FUNCTION_BLOCK ClearLinkMC EXTENDS FBA_TrifectaDrive IMPLEMENTS I_EncodedDrive
VAR_OUTPUT
	pulse AT %Q* : INT;
	brakeRelease AT %Q* : BOOL := TRUE;
	enable : BOOL;
	A : BOOL;
	B : BOOL;
	clear : BOOL;
END_VAR
VAR	
	hlfb AT %I* : REAL := -9999; //high level feedback, if -9999 then servo is idle
	
	outputRegister AT %Q* : INT;
	pulseRequest : INT;
	
	homingDelay : TON;
	resetPulse : TP;
	
	mode : (HOLD, TARGET, CONTINUOUS, RESET_ERR);
	calculation : (IDLE, DOWN, UP, CALCULATE, DONE);
	maxPosition : LREAL;
	
	position, targetPos : LREAL;
	
	pulsePosition : INT;
	pulseCounter : INT;
	rotationsPerPulse : INT; //revolutions per pulse
	displacementPerPulse : LREAL; //displacement per pulse
END_VAR
VAR_STAT CONSTANT
	resetWidth : TIME := T#500MS;
	delayWidth : TIME := T#500MS;
END_VAR
VAR //constructor
	homingDirectionOut : BOOL; 			//homing direction - see <A>
	minPosition : LREAL;
	displacementPerRotation : LREAL; 	//displacement per revolution	
	unitsPerPulse : INT := 800; 		//800 Teknic units per rotation - default setting is 800 units (1 rotation) per pulse
END_VAR

//M-connector output register
outputRegister.0 := enable AND bEnable; 	//enable
outputRegister.1 := A; 						//direction bit - T = outwards, F = inwards
outputRegister.2 := B; 						//homing bit - after startup, set to TRUE to begin homing, then set to FALSE to finish homing
outputRegister.3 := clear; 					//reset bit

rotationsPerPulse := unitsPerPulse/800; //Teknic constant - 800 units per rotation
displacementPerPulse := displacementPerRotation * rotationsPerPulse;

resetPulse(IN:= , PT:= resetWidth, Q=> clear, ET=> ); //reset pulse

IF NOT enable AND NOT AtInnerLimit THEN
	homingComplete := FALSE;
	step := Homing.IDLE;
	mode := HOLD;
END_IF

override();

CASE mode OF		
	HOLD: //hold current position, no motion
		pulse := 0;
		pulseRequest := 0;
	
	TARGET:	//target a given position
		
		IF WithinTolerance(position, targetPos, displacementPerPulse) THEN
			pulseRequest := 0;
			pulse := 0;
			mode := HOLD;
			
		ELSIF NOT Active THEN
			A :=  position < targetPos;
			(*
			2 options to traverse to a target position:
				a)  send all pulses at once - continuous motion but may exceed limits, check for bounds before setting
				b)  1 pulse at a time - choppy but safer
			*)
			targetPos := MAX(targetPos, minPosition); //if below minPosition, set to minPosition
			targetPos := MIN(targetPos, maxPosition); //if above maxPosition, set to maxPosition
			
			pulseRequest := TO_INT(ABS(position - targetPos)/displacementPerPulse);
			//pulseRequest := 1;
		END_IF
		
	CONTINUOUS: //single pulses in the direction specified by moveContinuous()
		pulseRequest := 1;
		
	RESET_ERR: //reset pulse, servo may need to be rehomed aftewards
		pulse := 0;
		pulseRequest := 0;
		resetPulse.IN := TRUE;
		
		IF resetPulse.Q THEN
			resetPulse.IN := FALSE;
			mode := HOLD;
		END_IF
		
END_CASE

sequence();

PROPERTY Active : BOOL
GET
Active := hlfb <> -9999;
END_GET
END_PROPERTY

{attribute 'monitoring':='call'}
PROPERTY AtOuterLimit : BOOL
GET
AtOuterLimit := outerLimit <> limitSensorDefaultState;
END_GET
END_PROPERTY

METHOD PRIVATE calculatePositions : BOOL
(*
the purpose of this method is calculate the position at the outer limit

complete a full range traverse while counting the pulses, then multiply
	displacement per rotation
	rotations per pulse
	number of pulses for the traversal
and add to position at inner limit to get position at outer limit
*)
CASE calculation OF
	IDLE:
		calculation := DOWN;
		
	DOWN:
		moveContinuous(direction := MC_Negative_Direction);
		IF AtInnerLimit THEN
			calculation := UP;
			pulseCounter := 0;
		END_IF
		
	UP:
		moveContinuous(direction := MC_Positive_Direction);
		IF AtHome THEN
			maxPosition := minPosition + (displacementPerRotation * rotationsPerPulse * pulseCounter);
			calculation := DONE;
		END_IF
		
	DONE:
		calculation := 0;
		calculatePositions := TRUE;
		
END_CASE
END_METHOD

PROPERTY CurrentPosition : LREAL
GET
CurrentPosition := position;

//CurrentPosition := pulsePosition * displacementPerPulse;
END_GET
SET
position := CurrentPosition;
END_SET
END_PROPERTY

PROPERTY Error : BOOL
GET
END_GET
END_PROPERTY

METHOD homingSequence : BOOL
homingDelay(IN:= , PT:= delayWidth, Q=> , ET=> );

CASE step OF
	Homing.IDLE:
		enable := TRUE;
		A := FALSE;
		B := TRUE;
		brakeRelease := TRUE;
		
		homingComplete := FALSE;
		
		homingDelay.IN := TRUE;
		IF homingDelay.Q THEN
			homingDelay.IN := FALSE;
			//step := Homing.START;
			step := Homing.RETRY;
		END_IF
		
	Homing.START:
		IF homingDelay.Q THEN
			homingDelay.IN := FALSE;
			step := Homing.SET;
			
		ELSIF AtHome THEN
			homingDelay.IN := TRUE;
			
		ELSIF AtOuterLimit THEN
			step := Homing.RETRY;
		
		ELSE
			enable := TRUE;
			A := FALSE;
			B := TRUE;
			brakeRelease := TRUE;
		
		END_IF
	
	Homing.RETRY:
		IF AtInnerLimit THEN
			homingDelay.IN := TRUE;
			enable := FALSE;
			
			IF homingDelay.Q THEN
				homingDelay.IN := FALSE;
				step := Homing.START;
			END_IF
			
		ELSE
			enable := TRUE;
			A := FALSE;
			B := FALSE;
			brakeRelease := TRUE;
			
			mode := CONTINUOUS;
		END_IF

	Homing.SET:
		enable := TRUE;
		A := FALSE;
		B := FALSE;
		brakeRelease := TRUE;
		
		IF calculatePositions() THEN
			step := Homing.DONE;
		END_IF
		
	Homing.DONE:
		homingSequence := homingComplete := TRUE;
		
		pulsePosition := 0;
		
		mode := HOLD;
		step := Homing.IDLE;
	
END_CASE
END_METHOD

{attribute 'TcRpcEnable'}
METHOD moveAbsolute : BOOL
VAR_INPUT
	newTarget : LREAL;
END_VAR
IF target >= maxPosition AND target <= minPosition THEN
	A :=  position < targetPos;
	targetPos := newTarget;
	mode := TARGET;
	
	moveAbsolute := TRUE;
END_IF
END_METHOD

{attribute 'TcRpcEnable'}
METHOD moveContinuous : BOOL
VAR_INPUT
	direction : MC_Direction;
END_VAR
IF direction = MC_Negative_Direction THEN
	A := FALSE;
ELSIF direction = MC_Positive_Direction THEN
	A := TRUE;
END_IF

mode := CONTINUOUS;
END_METHOD

{attribute 'TcRpcEnable'}
METHOD moveRelative : BOOL
VAR_INPUT
	distance : LREAL;
END_VAR
targetPos := targetPos + distance;

mode := TARGET;
END_METHOD

METHOD PRIVATE override : BOOL
VAR_INPUT
END_VAR
(*
allowable motion is between AtHome and AtInnerLimit
*)
IF AtHome AND NOT Active THEN
	IF homingDirectionOut THEN //homing is outwards
		position := maxPosition;
		pulsePosition := pulseCounter;
	ELSE
		position := minPosition;
		pulsePosition := 0;
	END_IF
	

ELSIF AtInnerLimit AND NOT Active THEN
	IF homingDirectionOut THEN //homing is outwards
		position := minPosition;
		pulsePosition := 0;
	ELSE
		position := maxPosition;
		pulsePosition := pulseCounter;
	END_IF
END_IF

CASE mode OF		
	HOLD:
		//
	
	TARGET:
		IF
			(AtHome AND TargetPosition > CurrentPosition) OR
			(AtInnerLimit AND TargetPosition > CurrentPosition) OR
			(AtOuterLimit AND TargetPosition < CurrentPosition)
		THEN
			mode := HOLD;
		END_IF
		
	CONTINUOUS:
		IF
			(AtHome AND A) OR
			(AtInnerLimit AND A) OR
			(AtOuterLimit AND NOT A)
		THEN
			mode := HOLD;
		END_IF
		
	RESET_ERR:
		//
		
END_CASE
END_METHOD

METHOD reset : BOOL
VAR_INPUT
END_VAR
mode := RESET_ERR;
END_METHOD

METHOD PRIVATE sequence : BOOL
VAR_INPUT
END_VAR
IF Active THEN //servo is active
	IF A THEN //positive direction
		position := position + (displacementPerPulse * pulse);
		pulsePosition := pulsePosition + pulse;
		
		pulseCounter := pulseCounter + pulse;
	ELSE //negative direction
		position := position - (displacementPerPulse * pulse);
		pulsePosition := pulsePosition - pulse;
		
		pulseCounter := pulseCounter - pulse;
	END_IF
	pulse := 0; //pulses already received, can be set to 0 so position change is not compounded

ELSIF pulse = 0 THEN //servo is not active
	pulse := pulseRequest;
END_IF

pulseRequest := 0; //remove this if not working as intended
END_METHOD

METHOD stop : BOOL
VAR_INPUT
END_VAR
mode := HOLD;
END_METHOD

PROPERTY TargetPosition : LREAL
GET
END_GET
SET
targetPos := TargetPosition;
END_SET
END_PROPERTY

METHOD toHome : BOOL
VAR_INPUT
END_VAR
IF homingDirectionOut THEN
	moveAbsolute(newTarget := maxPosition);
ELSE
	moveAbsolute(newTarget := minPosition);
END_IF
END_METHOD

END_FUNCTION_BLOCK

(* stored: Version 1.1.0.1, ProductVersion 3.1.4024.11
   POU ClearLinkMC: Id {c959ba26-8558-4921-981d-1da3c299d707}, SpecialFunc None
   Folder Private: Id {9b3fea93-f350-4628-abcc-bd49e2d7cd99}
   Folder Properties: Id {e78b63fe-cf71-47b5-ba6b-3023a80b30ce}
   Property Active: Id {807c9ae6-2791-4a9b-8015-1bf451a6a56b}
   Get Get: Id {aa4cc01a-37da-43cb-b30c-8e2bc563783d}
   Property AtOuterLimit: Id {6385a979-b10d-4caf-84a5-664acfc88266}
   Get Get: Id {eb0add8c-74bc-4bc2-93ab-6fcb2fc36408}
   Method calculatePositions: Id {e19e2a50-fb22-4fdb-a61a-d177c769d547}
   Property CurrentPosition: Id {75ebdd6d-7b75-4de5-8593-621bb72d6114}
   Get Get: Id {6856d05c-951f-4e2e-87df-ebd187d24ea1}
   Set Set: Id {1fda77e3-f52e-4259-845a-7410fc523da0}
   Property Error: Id {bda12f76-8849-4aa6-a93d-2a3f2d50597e}
   Get Get: Id {fa80b17b-fc29-4649-956e-d05d2b8946f1}
   Method homingSequence: Id {ab2757a4-d5f6-4f3f-addc-5f1377a21651}
   Method moveAbsolute: Id {50ef4f22-8da2-4b4e-8432-de0919b36ac2}
   Method moveContinuous: Id {6fae7e55-36e1-434b-b1d0-5392145a2ede}
   Method moveRelative: Id {a27e0a4f-4fbc-4d22-bb40-916e67eef58b}
   Method override: Id {c88d925b-2a9b-44f5-b155-07becad1ca73}
   Method reset: Id {148910f4-ce89-4537-a99c-bb0337253006}
   Method sequence: Id {a500267c-ac9c-4314-ade9-3f5adbe892a2}
   Method stop: Id {9c245f97-172f-4533-81f7-d28245b80a16}
   Property TargetPosition: Id {46ee9331-03d8-4e80-977f-3f6ec7fad893}
   Get Get: Id {c9bb5ba2-9737-4f8b-a18e-17d189211f37}
   Set Set: Id {b9e464bc-20f4-41e7-94ab-3937c1175ccd}
   Method toHome: Id {b88c291d-bab6-4c24-87c1-43e3a5206b24} *)
